FUNCTION_BLOCK basicEscalonamento (* Basic Function Block Type *)
  (* Standard: 61499-2 *)
  (* Version 0.0, 1/29/2026, Schneider Electric, Template *)
  PACKAGE Hidryco.HidrycoLib;
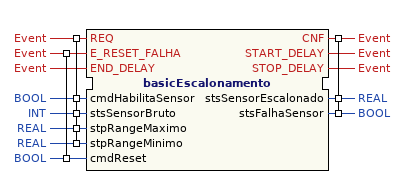
  EVENT_INPUT
    REQ WITH stsSensorBruto, cmdHabilitaSensor, stpRangeMaximo, stpRangeMinimo; (* Normal Execution Request *)
    E_RESET_FALHA WITH cmdReset;
    END_DELAY;
  END_EVENT
  EVENT_OUTPUT
    CNF WITH stsFalhaSensor, stsSensorEscalonado; (* Execution Confirmation *)
    START_DELAY;
    STOP_DELAY;
  END_EVENT
  VAR_INPUT
    cmdHabilitaSensor : BOOL;
    stsSensorBruto : INT; (* Input event qualifier *)
    stpRangeMaximo : REAL;
    stpRangeMinimo : REAL;
    cmdReset : BOOL;
  END_VAR
  VAR_OUTPUT
    stsSensorEscalonado : REAL;
    stsFalhaSensor : BOOL;
  END_VAR
  VAR
    bTimerAtivo : BOOL;
    bForaFaixa : BOOL;
    bFalhaAnt : BOOL;
    rValorAnt : REAL;
  END_VAR
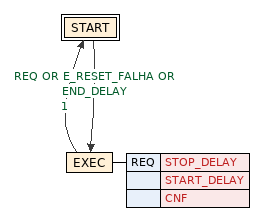
  EC_STATES
    START; (* Initial State *)
    EXEC : REQ -> STOP_DELAY, -> START_DELAY, -> CNF;
  END_STATES
  EC_TRANSITIONS
    START TO EXEC := REQ OR E_RESET_FALHA OR END_DELAY;
    EXEC TO START := 1;
  END_TRANSITIONS
  ALGORITHM REQ IN ST: (* Normally executed algorithm *)
(* ---- Zera eventos de saída: só sai o que for ligado abaixo ---- *)
STOP_DELAY  := FALSE;
START_DELAY := FALSE;
CNF         := FALSE;

bFalhaAnt := stsFalhaSensor;
rValorAnt := stsSensorEscalonado;

IF NOT cmdHabilitaSensor THEN
    (* ---- Sensor desabilitado: zera tudo ---- *)
    stsSensorEscalonado := 0.0;
    stsFalhaSensor      := FALSE;
    STOP_DELAY          := bTimerAtivo;
    bTimerAtivo         := FALSE;

ELSE
    (* ---- Sinal fora da faixa 4-20 mA ---- *)
    bForaFaixa := (stsSensorBruto < 3900) OR (stsSensorBruto > 20100);

    (* ---- Fim do tempo: confirma a falha se ainda fora ---- *)
    IF END_DELAY AND bTimerAtivo THEN
        bTimerAtivo := FALSE;
        IF bForaFaixa THEN
            stsFalhaSensor := TRUE;
        END_IF;
    END_IF;

    (* ---- Reset: só zera se o sinal já voltou à faixa ---- *)
    IF E_RESET_FALHA AND cmdReset AND stsFalhaSensor AND NOT bForaFaixa THEN
        stsFalhaSensor := FALSE;
    END_IF;

    (* ---- Temporizador ---- *)
    IF bForaFaixa AND NOT stsFalhaSensor AND NOT bTimerAtivo THEN
        START_DELAY := TRUE;        (* inicia contagem de 5 s *)
        bTimerAtivo := TRUE;
    ELSIF NOT bForaFaixa AND bTimerAtivo THEN
        STOP_DELAY  := TRUE;        (* sinal voltou: cancela *)
        bTimerAtivo := FALSE;
    END_IF;

    (* ---- Valor ---- *)
    IF stsFalhaSensor THEN
        stsSensorEscalonado := 0.0;
    ELSE
        stsSensorEscalonado := (INT_TO_REAL(stsSensorBruto) - 4000.0)
                               * (stpRangeMaximo - stpRangeMinimo) / 16000.0
                               + stpRangeMinimo;
        (* limita entre mínimo e máximo *)
        IF stpRangeMaximo >= stpRangeMinimo THEN
            IF stsSensorEscalonado < stpRangeMinimo THEN stsSensorEscalonado := stpRangeMinimo; END_IF;
            IF stsSensorEscalonado > stpRangeMaximo THEN stsSensorEscalonado := stpRangeMaximo; END_IF;
        ELSE
            IF stsSensorEscalonado > stpRangeMinimo THEN stsSensorEscalonado := stpRangeMinimo; END_IF;
            IF stsSensorEscalonado < stpRangeMaximo THEN stsSensorEscalonado := stpRangeMaximo; END_IF;
        END_IF;
    END_IF;
END_IF;

(* ---- Notifica só se mudou ---- *)
CNF := (stsSensorEscalonado <> rValorAnt) OR (stsFalhaSensor <> bFalhaAnt);
;
  END_ALGORITHM
END_FUNCTION_BLOCK
